# EPICS autosave request: acsMotionApp/Db/SPiiPlusCommut_settings.req
$(P)$(M):commut.VAL
